// TIA Portal V18 export
ORGANIZATION_BLOCK "Main"   // OB1, LAD, ProgramCycle
{ S7_Optimized_Access := 'TRUE' }
VERSION : 0.1
// stored: AutoNumber true, IsIECCheckEnabled false, SetENOAutomatically false
   VAR_INPUT
      Initial_Call : Bool;
      Remanence : Bool;
   END_VAR
   VAR_TEMP   // added for the SCL form of the ladder/FBD networks
      _w1 : Bool;
      _w2 : Bool;
      _w3 : Bool;
   END_VAR
BEGIN

REGION Network 1
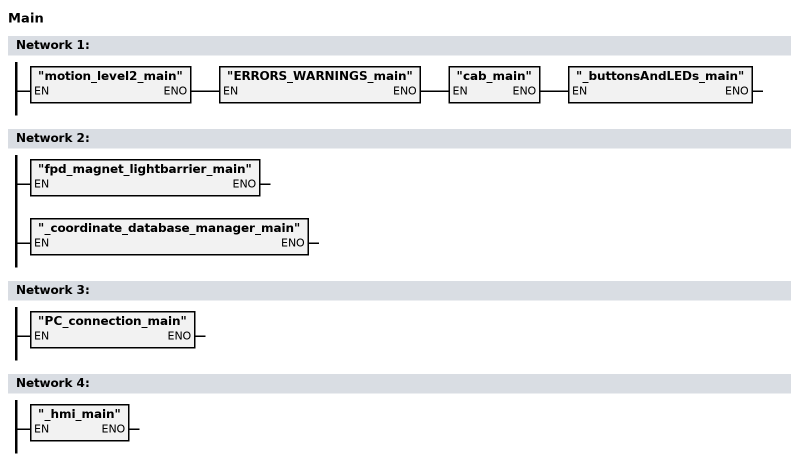
   RUNG wire#powerrail
      "motion_level2_main"()
      "ERRORS_WARNINGS_main"()
      "cab_main"()
      "_buttonsAndLEDs_main"()
   END_RUNG
   // the same network as SCL:
   "motion_level2_main"(ENO => #_w1);
   "ERRORS_WARNINGS_main"(EN := #_w1, ENO => #_w2);
   "cab_main"(EN := #_w2, ENO => #_w3);
   IF #_w3 THEN "_buttonsAndLEDs_main"(); END_IF;
END_REGION

REGION Network 2
   RUNG wire#powerrail
      "fpd_magnet_lightbarrier_main"()
   END_RUNG
   RUNG wire#powerrail
      "_coordinate_database_manager_main"()
   END_RUNG
   // the same network as SCL:
   "fpd_magnet_lightbarrier_main"();
   "_coordinate_database_manager_main"();
END_REGION

REGION Network 3
   RUNG wire#powerrail
      "PC_connection_main"()
   END_RUNG
   // the same network as SCL:
   "PC_connection_main"();
END_REGION

REGION Network 4
   RUNG wire#powerrail
      "_hmi_main"()
   END_RUNG
   // the same network as SCL:
   "_hmi_main"();
END_REGION
END_ORGANIZATION_BLOCK
